FUNCTION_BLOCK FB_mF_Test EXTENDS TcUnit.FB_TestSuite


valueShouldChangeWhenInputChanges();

METHOD valueShouldChangeWhenInputChanges
VAR
	mF : FB_mF;
	uTest : ARRAY[1..15] OF LREAL;
END_VAR

TEST('valueShouldChangeWhenInputChanges');
	uTest[1] := 5;
	mF.Step(
			u := uTest,
			y_meas := 2);
TEST_FINISHED();
END_METHOD

END_FUNCTION_BLOCK

(* stored: Version 1.1.0.1, ProductVersion 3.1.4024.9
   POU FB_mF_Test: Id {416b76a5-f41c-4a83-abf5-ec6ac421419b}, SpecialFunc None
   Method valueShouldChangeWhenInputChanges: Id {4ba9ccdb-35b9-4b07-8b9f-04437f83a946} *)
